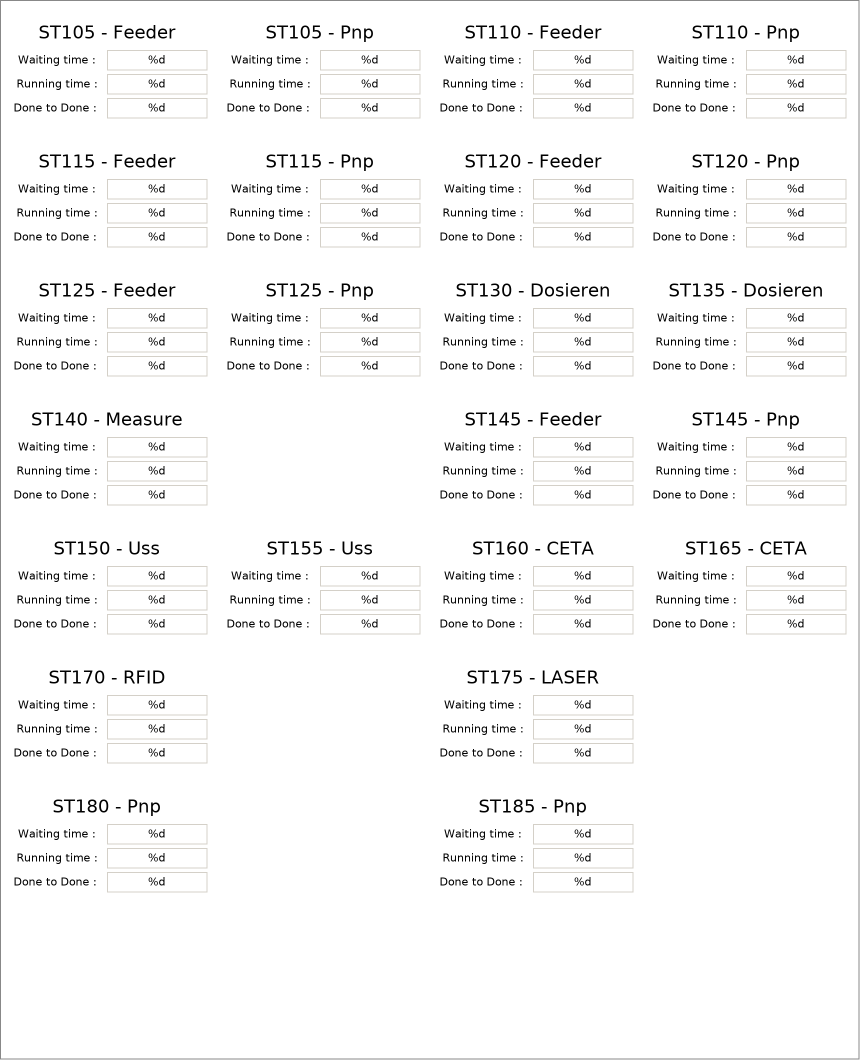
VISUALIZATION VISU_Time  // 860x1060
    Textfield (107,50 100x20), "%d", text variable: GVL.st105_aut.fb_stat_Feeder.tOUT_avgInWait_ms
    Label (7,50 100x20), "Waiting time :"
    Textfield (107,74 100x20), "%d", text variable: GVL.st105_aut.fb_stat_Feeder.tOUT_avgInRun_ms
    Label (7,74 100x20), "Running time :"
    Textfield (107,98 100x20), "%d", text variable: GVL.st105_aut.fb_stat_Feeder.tOUT_avgDoneToDone_ms
    Label (7,98 100x20), "Done to Done :"
    Label (7,19 200x27), "ST105 - Feeder"
    Textfield (320,50 100x20), "%d", text variable: GVL.st105_aut.fb_stat_pnp.tOUT_avgInWait_ms
    Label (220,50 100x20), "Waiting time :"
    Textfield (320,74 100x20), "%d", text variable: GVL.st105_aut.fb_stat_pnp.tOUT_avgInRun_ms
    Label (220,74 100x20), "Running time :"
    Textfield (320,98 100x20), "%d", text variable: GVL.st105_aut.fb_stat_pnp.tOUT_avgDoneToDone_ms
    Label (220,98 100x20), "Done to Done :"
    Label (220,19 200x27), "ST105 - Pnp"
    Textfield (533,50 100x20), "%d", text variable: GVL.st110_aut.fb_stat_Feeder.tOUT_avgInWait_ms
    Label (433,50 100x20), "Waiting time :"
    Textfield (533,74 100x20), "%d", text variable: GVL.st110_aut.fb_stat_Feeder.tOUT_avgInRun_ms
    Label (433,74 100x20), "Running time :"
    Textfield (533,98 100x20), "%d", text variable: GVL.st110_aut.fb_stat_Feeder.tOUT_avgDoneToDone_ms
    Label (433,98 100x20), "Done to Done :"
    Label (433,19 200x27), "ST110 - Feeder"
    Textfield (746,50 100x20), "%d", text variable: GVL.st110_aut.fb_stat_pnp.tOUT_avgInWait_ms
    Label (646,50 100x20), "Waiting time :"
    Textfield (746,74 100x20), "%d", text variable: GVL.st110_aut.fb_stat_pnp.tOUT_avgInRun_ms
    Label (646,74 100x20), "Running time :"
    Textfield (746,98 100x20), "%d", text variable: GVL.st110_aut.fb_stat_pnp.tOUT_avgDoneToDone_ms
    Label (646,98 100x20), "Done to Done :"
    Label (646,19 200x27), "ST110 - Pnp"
    Textfield (107,179 100x20), "%d", text variable: GVL.st115_aut.fb_stat_Feeder.tOUT_avgInWait_ms
    Label (7,179 100x20), "Waiting time :"
    Textfield (107,203 100x20), "%d", text variable: GVL.st115_aut.fb_stat_Feeder.tOUT_avgInRun_ms
    Label (7,203 100x20), "Running time :"
    Textfield (107,227 100x20), "%d", text variable: GVL.st115_aut.fb_stat_Feeder.tOUT_avgDoneToDone_ms
    Label (7,227 100x20), "Done to Done :"
    Label (7,148 200x27), "ST115 - Feeder"
    Textfield (320,179 100x20), "%d", text variable: GVL.st115_aut.fb_stat_pnp.tOUT_avgInWait_ms
    Label (220,179 100x20), "Waiting time :"
    Textfield (320,203 100x20), "%d", text variable: GVL.st115_aut.fb_stat_pnp.tOUT_avgInRun_ms
    Label (220,203 100x20), "Running time :"
    Textfield (320,227 100x20), "%d", text variable: GVL.st115_aut.fb_stat_pnp.tOUT_avgDoneToDone_ms
    Label (220,227 100x20), "Done to Done :"
    Label (220,148 200x27), "ST115 - Pnp"
    Textfield (533,179 100x20), "%d", text variable: GVL.st120_aut.fb_stat_Feeder.tOUT_avgInWait_ms
    Label (433,179 100x20), "Waiting time :"
    Textfield (533,203 100x20), "%d", text variable: GVL.st120_aut.fb_stat_Feeder.tOUT_avgInRun_ms
    Label (433,203 100x20), "Running time :"
    Textfield (533,227 100x20), "%d", text variable: GVL.st120_aut.fb_stat_Feeder.tOUT_avgDoneToDone_ms
    Label (433,227 100x20), "Done to Done :"
    Label (433,148 200x27), "ST120 - Feeder"
    Textfield (746,179 100x20), "%d", text variable: GVL.st120_aut.fb_stat_pnp.tOUT_avgInWait_ms
    Label (646,179 100x20), "Waiting time :"
    Textfield (746,203 100x20), "%d", text variable: GVL.st120_aut.fb_stat_pnp.tOUT_avgInRun_ms
    Label (646,203 100x20), "Running time :"
    Textfield (746,227 100x20), "%d", text variable: GVL.st120_aut.fb_stat_pnp.tOUT_avgDoneToDone_ms
    Label (646,227 100x20), "Done to Done :"
    Label (646,148 200x27), "ST120 - Pnp"
    Textfield (107,308 100x20), "%d", text variable: GVL.st125_aut.fb_stat_Feeder.tOUT_avgInWait_ms
    Label (7,308 100x20), "Waiting time :"
    Textfield (107,332 100x20), "%d", text variable: GVL.st125_aut.fb_stat_Feeder.tOUT_avgInRun_ms
    Label (7,332 100x20), "Running time :"
    Textfield (107,356 100x20), "%d", text variable: GVL.st125_aut.fb_stat_Feeder.tOUT_avgDoneToDone_ms
    Label (7,356 100x20), "Done to Done :"
    Label (7,277 200x27), "ST125 - Feeder"
    Textfield (320,308 100x20), "%d", text variable: GVL.st125_aut.fb_stat_pnp.tOUT_avgInWait_ms
    Label (220,308 100x20), "Waiting time :"
    Textfield (320,332 100x20), "%d", text variable: GVL.st125_aut.fb_stat_pnp.tOUT_avgInRun_ms
    Label (220,332 100x20), "Running time :"
    Textfield (320,356 100x20), "%d", text variable: GVL.st125_aut.fb_stat_pnp.tOUT_avgDoneToDone_ms
    Label (220,356 100x20), "Done to Done :"
    Label (220,277 200x27), "ST125 - Pnp"
    Textfield (533,308 100x20), "%d", text variable: GVL.st130_aut.fb_stat.tOUT_avgInWait_ms
    Label (433,308 100x20), "Waiting time :"
    Textfield (533,332 100x20), "%d", text variable: GVL.st130_aut.fb_stat.tOUT_avgInRun_ms
    Label (433,332 100x20), "Running time :"
    Textfield (533,356 100x20), "%d", text variable: GVL.st130_aut.fb_stat.tOUT_avgDoneToDone_ms
    Label (433,356 100x20), "Done to Done :"
    Label (433,277 200x27), "ST130 - Dosieren"
    Textfield (746,308 100x20), "%d", text variable: GVL.st135_aut.fb_stat.tOUT_avgInWait_ms
    Label (646,308 100x20), "Waiting time :"
    Textfield (746,332 100x20), "%d", text variable: GVL.st135_aut.fb_stat.tOUT_avgInRun_ms
    Label (646,332 100x20), "Running time :"
    Textfield (746,356 100x20), "%d", text variable: GVL.st135_aut.fb_stat.tOUT_avgDoneToDone_ms
    Label (646,356 100x20), "Done to Done :"
    Label (646,277 200x27), "ST135 - Dosieren"
    Textfield (107,437 100x20), "%d", text variable: GVL.st140_aut.fb_stat.tOUT_avgInWait_ms
    Label (7,437 100x20), "Waiting time :"
    Textfield (107,461 100x20), "%d", text variable: GVL.st140_aut.fb_stat.tOUT_avgInRun_ms
    Label (7,461 100x20), "Running time :"
    Textfield (107,485 100x20), "%d", text variable: GVL.st140_aut.fb_stat.tOUT_avgDoneToDone_ms
    Label (7,485 100x20), "Done to Done :"
    Label (7,406 200x27), "ST140 - Measure"
    Textfield (533,437 100x20), "%d", text variable: GVL.st145_aut.fb_stat_Feeder.tOUT_avgInWait_ms
    Label (433,437 100x20), "Waiting time :"
    Textfield (533,461 100x20), "%d", text variable: GVL.st145_aut.fb_stat_Feeder.tOUT_avgInRun_ms
    Label (433,461 100x20), "Running time :"
    Textfield (533,485 100x20), "%d", text variable: GVL.st145_aut.fb_stat_Feeder.tOUT_avgDoneToDone_ms
    Label (433,485 100x20), "Done to Done :"
    Label (433,406 200x27), "ST145 - Feeder"
    Textfield (746,437 100x20), "%d", text variable: GVL.st145_aut.fb_stat_pnp.tOUT_avgInWait_ms
    Label (646,437 100x20), "Waiting time :"
    Textfield (746,461 100x20), "%d", text variable: GVL.st145_aut.fb_stat_pnp.tOUT_avgInRun_ms
    Label (646,461 100x20), "Running time :"
    Textfield (746,485 100x20), "%d", text variable: GVL.st145_aut.fb_stat_pnp.tOUT_avgDoneToDone_ms
    Label (646,485 100x20), "Done to Done :"
    Label (646,406 200x27), "ST145 - Pnp"
    Textfield (107,566 100x20), "%d", text variable: GVL.st150_aut.fb_stat.tOUT_avgInWait_ms
    Label (7,566 100x20), "Waiting time :"
    Textfield (107,590 100x20), "%d", text variable: GVL.st150_aut.fb_stat.tOUT_avgInRun_ms
    Label (7,590 100x20), "Running time :"
    Textfield (107,614 100x20), "%d", text variable: GVL.st150_aut.fb_stat.tOUT_avgDoneToDone_ms
    Label (7,614 100x20), "Done to Done :"
    Label (7,535 200x27), "ST150 - Uss"
    Textfield (320,566 100x20), "%d", text variable: GVL.st155_aut.fb_stat.tOUT_avgInWait_ms
    Label (220,566 100x20), "Waiting time :"
    Textfield (320,590 100x20), "%d", text variable: GVL.st155_aut.fb_stat.tOUT_avgInRun_ms
    Label (220,590 100x20), "Running time :"
    Textfield (320,614 100x20), "%d", text variable: GVL.st155_aut.fb_stat.tOUT_avgDoneToDone_ms
    Label (220,614 100x20), "Done to Done :"
    Label (220,535 200x27), "ST155 - Uss"
    Textfield (533,566 100x20), "%d", text variable: GVL.st160_aut.fb_stat.tOUT_avgInWait_ms
    Label (433,566 100x20), "Waiting time :"
    Textfield (533,590 100x20), "%d", text variable: GVL.st160_aut.fb_stat.tOUT_avgInRun_ms
    Label (433,590 100x20), "Running time :"
    Textfield (533,614 100x20), "%d", text variable: GVL.st160_aut.fb_stat.tOUT_avgDoneToDone_ms
    Label (433,614 100x20), "Done to Done :"
    Label (433,535 200x27), "ST160 - CETA"
    Textfield (746,566 100x20), "%d", text variable: GVL.st165_aut.fb_stat.tOUT_avgInWait_ms
    Label (646,566 100x20), "Waiting time :"
    Textfield (746,590 100x20), "%d", text variable: GVL.st165_aut.fb_stat.tOUT_avgInRun_ms
    Label (646,590 100x20), "Running time :"
    Textfield (746,614 100x20), "%d", text variable: GVL.st165_aut.fb_stat.tOUT_avgDoneToDone_ms
    Label (646,614 100x20), "Done to Done :"
    Label (646,535 200x27), "ST165 - CETA"
    Textfield (107,695 100x20), "%d", text variable: GVL.st170_aut.fb_stat.tOUT_avgInWait_ms
    Label (7,695 100x20), "Waiting time :"
    Textfield (107,719 100x20), "%d", text variable: GVL.st170_aut.fb_stat.tOUT_avgInRun_ms
    Label (7,719 100x20), "Running time :"
    Textfield (107,743 100x20), "%d", text variable: GVL.st170_aut.fb_stat.tOUT_avgDoneToDone_ms
    Label (7,743 100x20), "Done to Done :"
    Label (7,664 200x27), "ST170 - RFID"
    Textfield (533,695 100x20), "%d", text variable: GVL.st175_aut.fb_stat.tOUT_avgInWait_ms
    Label (433,695 100x20), "Waiting time :"
    Textfield (533,719 100x20), "%d", text variable: GVL.st175_aut.fb_stat.tOUT_avgInRun_ms
    Label (433,719 100x20), "Running time :"
    Textfield (533,743 100x20), "%d", text variable: GVL.st175_aut.fb_stat.tOUT_avgDoneToDone_ms
    Label (433,743 100x20), "Done to Done :"
    Label (433,664 200x27), "ST175 - LASER"
    Textfield (107,824 100x20), "%d", text variable: GVL.st180_aut.fb_stat.tOUT_avgInWait_ms
    Label (7,824 100x20), "Waiting time :"
    Textfield (107,848 100x20), "%d", text variable: GVL.st180_aut.fb_stat.tOUT_avgInRun_ms
    Label (7,848 100x20), "Running time :"
    Textfield (107,872 100x20), "%d", text variable: GVL.st180_aut.fb_stat.tOUT_avgDoneToDone_ms
    Label (7,872 100x20), "Done to Done :"
    Label (7,793 200x27), "ST180 - Pnp"
    Textfield (533,824 100x20), "%d", text variable: GVL.st185_aut.fb_stat.tOUT_avgInWait_ms
    Label (433,824 100x20), "Waiting time :"
    Textfield (533,848 100x20), "%d", text variable: GVL.st185_aut.fb_stat.tOUT_avgInRun_ms
    Label (433,848 100x20), "Running time :"
    Textfield (533,872 100x20), "%d", text variable: GVL.st185_aut.fb_stat.tOUT_avgDoneToDone_ms
    Label (433,872 100x20), "Done to Done :"
    Label (433,793 200x27), "ST185 - Pnp"
END_VISUALIZATION

(* stored: Version 1.1.0.1, ProductVersion 3.1.4024.6
   Visu VISU_Time: Id {edb4d9db-d2bd-4547-ad5a-562ace8339d4} *)
